// Function block for EtherCAT diagnosis, looking at the live slave status and reporting back any missing slaves
FUNCTION_BLOCK FB_EthercatDiagnosis IMPLEMENTS I_EthercatDiagnosis
VAR
	_ignoredSlaves	: ARRAY[0..Tc2_EtherCAT.EC_MAX_SLAVES] OF Tc2_System.T_MaxString;
	_missingSlaves	: ARRAY[0..Tc2_EtherCAT.EC_MAX_SLAVES] OF ST_EthercatSlaveInfo;
	_status			: E_EthercatDiagnosisStatus;
	_diagState		: E_EthercatDiagnosisState;
	_error			: BOOL;
END_VAR

(* Returns TRUE if an error occurred while performing the scan*)
PROPERTY Error : BOOL
GET
Error := _error;
END_GET
END_PROPERTY

(* Gets an array of slaves that have been added to ignore list*)
PROPERTY IgnoredSlaves : REFERENCE TO ARRAY [0..Tc2_EtherCAT.EC_MAX_SLAVES] OF Tc2_System.T_MaxString
GET
IgnoredSlaves REF= _ignoredSlaves;
END_GET
END_PROPERTY

{warning 'add method implementation '}
(* Adds the provided slave to a collection of slaves that will not trigger an error
 Example is slaves that are used on hot connect groups, and when connected should not cause an error. *)
METHOD IgnoreSlave
VAR_INPUT
	(* Slave to be ignored if not found or an error is reported back*)
	name	: Tc2_System.T_MaxString;
END_VAR
IF name <> '' THEN
	ArrayHelper.InsertAtStart(arr := _ignoredSlaves, item := name);
END_IF
END_METHOD

(* Returns an array of misisng slave names*)
PROPERTY MissingSlaves : REFERENCE TO ARRAY [0..Tc2_EtherCAT.EC_MAX_SLAVES] OF ST_EthercatSlaveInfo
GET
MissingSlaves REF= _missingSlaves;
END_GET
END_PROPERTY

{warning 'add method implementation '}
(* Reset the internal state machine of diagnosis and clearing any errors, if active.*)
METHOD Reset
END_METHOD

{warning 'add method implementation '}
(* Performs a scan on the EtherCAT master, returns TRUE when done.*)
METHOD Scan : BOOL
VAR_INPUT
	EcMasterNetId	: AMSNETID;
END_VAR
END_METHOD

(* Gets the status based on last executed scan.*)
PROPERTY Status : E_EthercatDiagnosisStatus
GET
Status := _status;
END_GET
END_PROPERTY

END_FUNCTION_BLOCK

(* stored: Version 1.1.0.1, ProductVersion 3.1.4024.14
   POU FB_EthercatDiagnosis: Id {d33d9930-1765-079a-0b49-5f9960a4f2c8}, SpecialFunc None
   Property Error: Id {1a117e49-56cb-0db0-21bf-7dac4cb52b82}
   Get Get: Id {bf5b31d6-0b1e-07d4-0303-b362fefe22c3}
   Property IgnoredSlaves: Id {7608aaf4-3882-00d8-3f05-e8979b4d9600}
   Get Get: Id {d9f798d0-70ea-0ed9-1bdf-e9314e35a335}
   Method IgnoreSlave: Id {42e52eac-60a4-0644-0bec-21bc97b0aa37}
   Property MissingSlaves: Id {b9124aca-eb02-0db3-3a56-63cbcceec356}
   Get Get: Id {db0dc646-f425-0868-2335-14eb7fab3a9f}
   Method Reset: Id {e45d3a11-10d1-08d9-0251-149985ae99a8}
   Method Scan: Id {1773b74b-9cad-0138-159e-d607f5ab1800}
   Property Status: Id {9ef092d6-a48c-0b76-06a8-af961e0ab80a}
   Get Get: Id {b87cbbbe-6dbc-0b5d-16fb-f14ec525857d} *)
